//==================================================================================================
//							Beckhoff Automation Poland
//									18.04.2018
//	Struktura zawierajaca I/O odpowiedniego bloku
//  v1.0	|| TC v 3.1.4022.16		|| - pierwsza wersja
//==================================================================================================
TYPE ST_MCHaltIO:
STRUCT
	bExecute						: BOOL;								// Rising edge executes cmd
	lrDeceleration					: LREAL;
	lrJerk							: LREAL;
	eBufferMode						: Tc2_MC2.MC_BufferMode;
	stOptions						: Tc2_MC2.ST_MoveOptions;
	bDone							: BOOL;
	bBusy							: BOOL;
	bActive							: BOOL;
	bCommandAborted					: BOOL;
	bError							: BOOL;
	udiErrorID						: UDINT;
END_STRUCT
END_TYPE

(* stored: Version 1.1.0.1, ProductVersion 3.1.4026.13, FileIdentifier 0c5c000b13766b1b7b7b995b6f00f7072766f884, FileSignature 4eadb95fe7216fee295790dcc8288618695cf059f7ea2aa752c6d8544af0b89a7832ec1a04e81d90dd5168130b84657317131e3b8bdf530d2e26ad3c9b68769422099e354afbef72a649b7a336698111c677ea57902a51c21c4920e6e99f3395585bd68fc700bb14a80360aa42741937c350479afdfe8dcc70c5a7fd5fc79a2a907bf50426abcb64dc0f442ac0d63c7cb594a788ccf1a2590f3ae6d9aa923183d7cb905af0cb8425b4465271a1ff5da5cef3d2afdf67d02bbe73670bbeb24ca32e7d9239687ba672baa7b68ef940bacf60e8b0b7c149a0ee01983bdf88b6c4c6c5bf3c9a0aff66113bd5f149ffa9735090fb6414041b8c1fcfb6af3bbd1596d1
   DUT ST_MCHaltIO: Id {a449ec57-5115-45df-b66f-f74e3de84fab} *)
